Staubli VAL3: _stopCycle.pjx

--- _stopCycle.pjx ---
Parameters version=s7.7 stackSize=5000 millimeterUnit=true
Program file=start.pgx
Program file=stop.pgx
Data file=_stopCycle.dtx
Library alias=cycleStatus path=Disk://cycleStatus/cycleStatus.pjx

--- start.pgx ---
program start()
begin
  // stop Cycle
  cycleStatus:bToStop=true
  watch(cycleStatus:bToStop==false,1)
end
